FUNCTION_BLOCK FB_CTUD_UDINT (* Up Down counter (UDINT) *)
  (* Standard: 61499-1; Description: Copyright (c) 2023 Martin Erich Jobst This program and the accompanying materials are made available under the terms of the Eclipse Public License 2.0 which is available at https://www.eclipse.org/legal/epl-2.0/ SPDX-License-Identifier: EPL-2.0 Some portions generated by Gemini CLI *)
  (* Version 3.1, 2026-02-01, Franz Höpfinger, HR Agrartechnik GmbH, copy from ULINT and made UDINT *)
  (* Version 3.0, 2025-04-14, Patrick Aigner, changed package *)
  (* Version 1.0, 2023-04-28, Martin Jobst *)
  PACKAGE iec61131::counters;
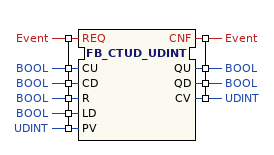
  EVENT_INPUT
    REQ WITH CU, CD, R, LD, PV; (* Normal Execution Request *)
  END_EVENT
  EVENT_OUTPUT
    CNF WITH QU, QD, CV; (* Execution Confirmation *)
  END_EVENT
  VAR_INPUT
    CU : BOOL; (* Count up *)
    CD : BOOL; (* Count down *)
    R : BOOL; (* Reset *)
    LD : BOOL; (* Load *)
    PV : UDINT; (* Preset value *)
  END_VAR
  VAR_OUTPUT
    QU : BOOL; (* Output up *)
    QD : BOOL; (* Output down *)
    CV : UDINT; (* Count value *)
  END_VAR
  EC_STATES
    REQ : REQ -> CNF;
  END_STATES
  ALGORITHM REQ IN ST:
IF R THEN
	CV := 0;
ELSE
	IF LD THEN
		CV := PV;
	ELSE
		IF NOT (CU AND CD) THEN
			IF CU AND CV < 4294967295 THEN
				CV := CV + 1;
			ELSIF CD AND CV > 0 THEN
				CV := CV - 1;
			END_IF;
		END_IF;
	END_IF;
END_IF;
QU := CV >= PV;
QD := CV <= 0;
  END_ALGORITHM
END_FUNCTION_BLOCK
